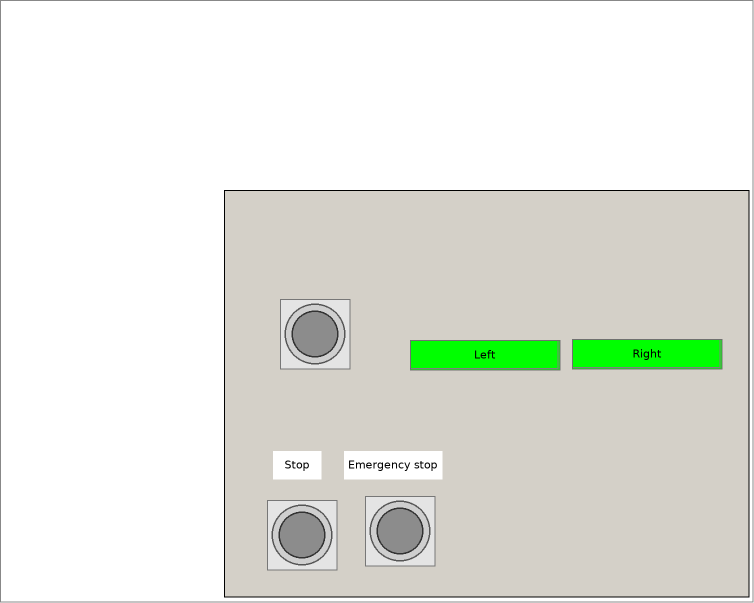
VISUALIZATION HMI  // 754x603
    Rectangle (224,190 525x407)
    Polyline (573,328)
    PushSwitch (267,500 70x70), variable: Stop.Stop_Button, behaviour: TAP, style: Switch-PushSwitch-Gray
    PushSwitch (365,496 70x70), variable: Emergency_Stop.Stop_Button, behaviour: TAP, style: Switch-PushSwitch-Gray
    Button (410,340 150x30), "Left", colour toggle: GVL.qxGotoPosA
        tap Manual.Left
    Button (572,339 150x30), "Right", colour toggle: GVL.qxGotoPosB
        tap Manual.Right
    Textfield (272,450 50x30), "Stop"
    Textfield (343,450 100x30), "Emergency stop"
    PushSwitchLed (280,299 70x70), variable: Automatic_Or_Manual.Automatic_Or_Manual, invisible if: MAIN.Visible, behaviour: TOGGLE, style: Switch-PushSwitchLed-Gray
END_VISUALIZATION

(* stored: Version 1.1.0.1, ProductVersion 3.1.4024.12
   Visu HMI: Id {d4fdea4d-848a-4d81-afe3-55505be43d78} *)
